FUNCTION_BLOCK E_SWITCH (* Switch(demultiplex)an event *)
  (* Standard: 61499-1; Classification: Event Processing; Function: Event Switch *)
  (* Version 0.1, 2003-12-30, JHC, Rockwell Automation, Updated for 61499-1 CDV. *)
  (* Version 0.0, 2001-04-14, JHC, Rockwell Automation, First XML version. *)
  (* Compiler header: package fb.rt.events; *)
  (* Compiler Java IBM VisualAge 3.0 *)
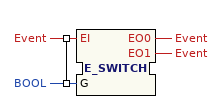
  EVENT_INPUT
    EI WITH G; (* Event Input *)
  END_EVENT
  EVENT_OUTPUT
    EO0; (* Output,switched from EI when G=0 *)
    EO1; (* Output,switched from EI when G=1 *)
  END_EVENT
  VAR_INPUT
    G : BOOL; (* Switch EI to EI0 when G=0,to EI1 when G=1 *)
  END_VAR
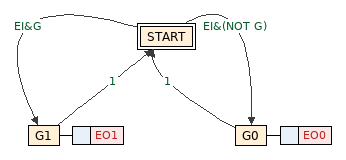
  EC_STATES
    START; (* Initial State *)
    G0 : -> EO0; (* Issue EO0 when EI arrives with G=0 *)
    G1 : -> EO1; (* Issue EO1 when EI arrives with G=1 *)
  END_STATES
  EC_TRANSITIONS
    START TO G0 := EI&(NOT G);
    G0 TO START := 1;
    START TO G1 := EI&G;
    G1 TO START := 1;
  END_TRANSITIONS
END_FUNCTION_BLOCK
